TEXTLIST AUTOMATA_lepesek1
  0 = 'Készenléti állapot'
  1 = 'Várakozás az NTC vágóra'
  2 = 'A szán indítása'
  3 = 'A szán az előhajlítóhoz mozog...'
  4 = 'Előhajlítás...'
  5 = 'Véghajlításhoz indul'
  6 = 'A szán a véghajlításhoz mozog...'
  7 = 'Véghajlítás indítása'
  8 = 'Véghajlítás...'
  9 = 'A szán indítása'
  10 = '1. hegesztés, várakozás a szánra'
  11 = '1. hegesztés, fej indítása'
  12 = '1. hegesztés, várakozás a fejre'
  13 = '1. hegesztés folyamatban...'
  14 = '1. hegesztés, fej vissza'
  15 = '1. hegesztés, fej vissza'
  16 = '3. hegesztés, várakozás a szánra'
  17 = '3. hegesztés, fej indítása'
  18 = '3. hegesztés, várakozás a fejre'
  19 = '3. hegesztés, hegesztés folyamatban'
  20 = '3. hegesztés, fej vissza'
  21 = '3. hegesztés, fej vissza'
  22 = '2. hegesztés, várakozás a szánra'
  23 = '2. hegesztés, fej indítása'
  24 = '2. hegesztés, várakozás a fejre'
  25 = '2. hegesztés, hegesztés folyamatban'
  26 = '2. hegesztés, fej vissza'
  27 = '2. hegesztés, fej vissza'
  28 = '4. hegesztés, várakozás a szánra'
  29 = 'Várakozás az NTC vágás végére'
  30 = 'Várakozás a robotra'
  31 = 'A robot az NTC-ért megy'
  32 = 'A robot az NTC-ért megy'
  33 = 'Várakozás az NTC elengedésére'
  34 = 'A robot az NTC-t a 4. hegesztéshez viszi'
  35 = '4. hegesztés, fej indítása'
  36 = '4. hegesztés, várakozás a fejre'
  37 = '4. hegesztés, hegesztés folyamatban'
  38 = '4. hegesztés, fej vissza'
  39 = '4. hegesztés, fej vissza'
  40 = '4. hegesztés, robot elmegy'
  41 = '4. hegesztés, robot elmegy'
  42 = '5. hegesztés, várakozás a szánra'
  43 = '5. hegesztés, fej indítása'
  44 = '5. hegesztés, várakozás a fejre'
  45 = '5. hegesztés, hegesztés folyamatban'
  46 = '5. hegesztés, fej vissza'
  47 = '5. hegesztés, fej vissza'
  48 = 'A szán indítása'
  49 = 'A szán a kamerás ellenörzéshez mozog...'
  50 = 'Kamerás végértékelés'
  60 = 'A szán a kamerás ellenörzéshez mozog...'
  61 = 'Betett termék kamerás ellenörzése'
  62 = 'A szán indítása'
  99 = 'STOP utáni várakozás'
  100 = 'A szán indítása a szervízboxhoz'
  101 = 'Szervízbox, várakozás a szánra'
  102 = 'Várakozás az adapter\nkivételére'
  103 = 'Várakozás az adapter\nkivétele után'
  105 = 'Várakozás...'
  110 = 'NTC vágó ellenörzése'
  111 = 'Döntés új NTC vágásról'
  112 = 'Várakozás az NTC vágóra'
  113 = 'Várakozás az NTC megfogó nyitására'
  120 = 'Termék berakás, megigazítás'
  121 = 'Várakozás a folytatásra'
  130 = 'NTC tengely leállítása'
  131 = 'Hegesztöfejek visszahúzása'
  132 = 'Várakozás a hegesztöfejek\nvisszahúzódására'
  133 = 'Robot pozíció ellenörzése'
  134 = 'Robot HOME-ba érkezésére vár'
  135 = 'Várakozás a hajlító- és\nhegesztöfejek visszahúzódására'
  140 = '1. hegesztöfej visszahúzása'
  141 = 'Várakozás az 1. hegesztőfej\nvisszahúzódására'
  142 = 'Várakozás a szán szervízboxba\n\nérkezésére'
  143 = 'Várakozás a folytatásra'
  150 = '1. hegesztöfej visszahúzása'
  151 = 'Várakozás az 1. hegesztőfej\nvisszahúzódására'
  152 = 'Várakozás a szán szervízboxba\n\nérkezésére'
  153 = 'Várakozás a folytatásra'
  160 = '1. hegesztöfej visszahúzása'
  161 = 'Várakozás az 1. hegesztőfej\nvisszahúzódására'
  162 = 'Várakozás a szán szervízboxba\n\nérkezésére'
  163 = 'Várakozás a folytatásra'
  170 = '2. hegesztöfej visszahúzása'
  171 = 'Várakozás az 2. hegesztőfej\nvisszahúzódására'
  172 = 'Várakozás a folytatásra'
  180 = '2. hegesztöfej visszahúzása'
  181 = 'Várakozás az 2. hegesztőfej\nvisszahúzódására'
  182 = 'Várakozás a szán szervízboxba\n\nérkezésére'
  183 = 'Várakozás a folytatásra'
  190 = 'Adapter pótlólagos felhelyezése, munkadarab rögzítése'
  300 = 'NTC oldali folyamat felfüggesztve'
   = ''
END_TEXTLIST

(* stored: Version 1.1.0.1, ProductVersion 3.1.4020.3
   TextList AUTOMATA_lepesek1: Id {173280f2-ebd2-4baa-9cbb-3710d3f7135d} *)
